FUNCTION F_ITC_SendRAC : BOOL
(**************************************************************************************
 * 	Application		:	BoxControl Framework
 *	Revision		:	$Revision: 404529 $
 *	Revision date	:	$Date: 2018-04-23 08:21:38 +0200 (Mo., 23 Apr 2018) $
 *	Last changed by	:	$Author: b7bolm $
 *	URL				:	$URL: http://almscdc.swisslog.com/repo/SWPD/Development/BoxControlFramework/20_Release/trunk/01_Software/BCF/BCF/JumpStart/20_Product/10_App/11_Com/10_Lib/10_Conv/11_ITC/F_ITC_SendRAC.TcPOU $
 *
 *	Purpose			:	Wrap message - RAC
 *
 * ------------------------------------------------------------------------------------
 *	Copyright Swisslog [IP AG], Switzerland. All rights reserved.
 * 
 * ------------------------------------------------------------------------------------
 *	
 * 	Revision History: 
 *
 * 	VERSION			DATE			INITIALS			DESCRIPTION
 *	0.1				01.01.2001		swl					Example
 *
 **************************************************************************************)
VAR_INPUT
	eChannelSrc				: E_MFCS_Channel; // Source communicaton channel
	PositionName			: STRING(Conveyor.POSITION_STRINGLENGTH); // SIS MM-GGG-EEEE-FF-Z
	CommandDataIndex		: INT;
	AssignmentID			: UDINT;
	GroupID					: ULINT;
	eReturnCode				: E_ErrorConv; // Return code
END_VAR
VAR
	RAC						: ST_ITC_RAC; 
END_VAR

// Map values
RAC.Position := PositionName;
RAC.CommandDataIndex := CommandDataIndex;
RAC.AssignmentID := AssignmentID;
RAC.GroupID := GroupID;
RAC.eReturnCode := eReturnCode;

// Forward to ITC
F_ITC_SendRAC := fbITC_Manager.M_SendData(
					meChannel	:= eChannelSrc,
					mMsgType	:= E_ITC_MsgTypeConv.ROBOT_ACTION_COMPLETE,
					mpData		:= ADR(RAC),
					mLen		:= SIZEOF(RAC));

END_FUNCTION

(* stored: Version 1.1.0.1, ProductVersion 3.1.4022.12
   POU F_ITC_SendRAC: Id {cd94148f-e04d-441d-a058-51627bde7a63}, SpecialFunc None *)
